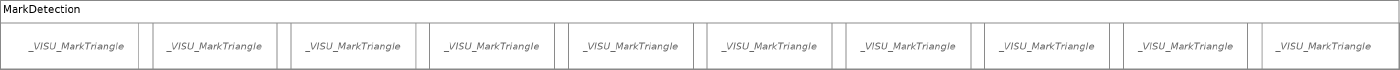
VISUALIZATION _VISU_MarkDefinition_View_edit  // 1463x74
VAR_IN_OUT
	mInst : FB_MarkDefinition;
  xScale : UDINT;
END_VAR
    Frame (0,24 160x50), invisible if: NOT mInst.sMarkDef[1].bShow
        shows _VISU_MarkTriangle(mInst := mInst.sMarkDef[1])
    Frame (144,24 160x50), invisible if: NOT mInst.sMarkDef[2].bShow
        shows _VISU_MarkTriangle(mInst := mInst.sMarkDef[2])
    Frame (289,24 160x50), invisible if: NOT mInst.sMarkDef[3].bShow
        shows _VISU_MarkTriangle(mInst := mInst.sMarkDef[3])
    Frame (724,24 160x50), invisible if: NOT mInst.sMarkDef[6].bShow
        shows _VISU_MarkTriangle(mInst := mInst.sMarkDef[6])
    Frame (434,24 160x50), invisible if: NOT mInst.sMarkDef[4].bShow
        shows _VISU_MarkTriangle(mInst := mInst.sMarkDef[4])
    Frame (579,24 160x50), invisible if: NOT mInst.sMarkDef[5].bShow
        shows _VISU_MarkTriangle(mInst := mInst.sMarkDef[5])
    Frame (869,24 160x50), invisible if: NOT mInst.sMarkDef[7].bShow
        shows _VISU_MarkTriangle(mInst := mInst.sMarkDef[7])
    Frame (1303,24 160x50), invisible if: NOT mInst.sMarkDef[10].bShow
        shows _VISU_MarkTriangle(mInst := mInst.sMarkDef[10])
    Frame (1014,24 160x50), invisible if: NOT mInst.sMarkDef[8].bShow
        shows _VISU_MarkTriangle(mInst := mInst.sMarkDef[8])
    Frame (1159,24 160x50), invisible if: NOT mInst.sMarkDef[9].bShow
        shows _VISU_MarkTriangle(mInst := mInst.sMarkDef[9])
    Rectangle (0,0 120x20), "MarkDetection"
END_VISUALIZATION

(* stored: Version 1.1.0.1, ProductVersion 3.1.4024.11
   Visu _VISU_MarkDefinition_View_edit: Id {d4efe329-2415-42c5-9647-e9134db2d461} *)
